// TwinCAT 3 PLC project TrafficLightTests
// ProgramVersion: 3.1.4026.22
// libraries:
//   Tc2_Standard, * (Beckhoff Automation GmbH)
//   Tc2_System, * (Beckhoff Automation GmbH)
//   TcUnit, * (www.tcunit.org)
//   B3TrafficLight_Plc,newest,Tc3 Project
// project tree:
//   / PlcTask.TcTTO
//   POUs/ FB_TrafficLightConsumer.TcPOU, MAIN.TcPOU
// (motion and I/O tree: see PLC project b3trafficlight_plc)

CONFIGURATION TrafficLightTests
    RESOURCE PLC ON TwinCAT3
        TASK PlcTask(INTERVAL := T#10ms, PRIORITY := 21);
        PROGRAM MAIN WITH PlcTask : MAIN;
    END_RESOURCE
END_CONFIGURATION

// ---- POUs/MAIN.TcPOU
PROGRAM MAIN
VAR
END_VAR

END_PROGRAM

// ---- POUs/FB_TrafficLightConsumer.TcPOU
FUNCTION_BLOCK FB_TrafficLightConsumer
VAR
    light : B3TrafficLight_Plc.FB_TrafficLight;
    lastState : INT;
END_VAR

lastState := light.Step();

END_FUNCTION_BLOCK
